TYPE ST_Point :
STRUCT
	x : LREAL;
	y : LREAL;
END_STRUCT
END_TYPE

(* stored: Version 1.1.0.1, ProductVersion 3.1.4024.12
   DUT ST_Point: Id {c7225085-c2e5-4554-8b0c-221de5a7bfd6} *)
